// TIA Portal V17 export
// export: Created 2024-08-09T12:53:14.745239Z, ExportSetting WithDefaults, DisplayName Totally Integrated Automation Portal, DisplayVersion V17 Update 7, DisplayName TIA Portal Openness, DisplayVersion V17 Update 7, DisplayName TIA Portal Version Control Interface, DisplayVersion V17, DisplayName STEP 7 Professional, DisplayVersion V17 Update 7, DisplayName STEP 7 Safety, DisplayVersion V17 Update 6, DisplayName WinCC Professional, DisplayVersion V17 Update 7
VAR_GLOBAL   // PLC tag table "Dec_Niveaux_TRANSF"
END_VAR
VAR_GLOBAL CONSTANT   // user constants
   TRANSF_Repos_Niv : USInt := 0;
   TRANSF_AttenteAval_Niv : USInt := 15;
   TRANSF_AttenteAmont_Niv : USInt := 30;
   TRANSF_Lancement_Niv : USInt := 45;
   TRANSF_Prepositionnement_Niv : USInt := 60;
   TRANSF_AttenteCircuitPositionne_Niv : USInt := 75;
   TRANSF_AttenteProduit_Niv : USInt := 90;
   TRANSF_Surveillance_Niv : USInt := 105;
   TRANSF_ChangementDestination_Niv : USInt := 165;
   TRANSF_Vidange_Niv : USInt := 195;
   TRANSF_MajBase_Niv : USInt := 210;
   TRANSF_FinLot_Niv : USInt := 255;
   TRANSF_ChangementNoeud_Niv : USInt := 180;
   TRANSF_DefOrigine_Niv : USInt := 120;
   TRANSF_ArretSource_Niv : USInt := 150;
   TRANSF_Suspension_Niv : USInt := 135;
END_VAR
